SUBAPPLICATION I_GetAttribute_IDA (* Bündelung von I_GetAttribute (Kommando GetAttribute F.58) und Attribute_IDA (asynchroner Adapter-Empfang) mit gemeinsamen u16ObjId und u8AID Parametern *)
  (* Standard: 61499-2; Description: Copyright (c) 2026 Meisterschulen am Ostbahnhof This program and the accompanying materials are made available under the terms of the Eclipse Public License 2.0 which is available at https://www.eclipse.org/legal/epl-2.0/ SPDX-License-Identifier: EPL-2.0 *)
  (* Version 1.0, 2026-09-15, Franz Höpfinger, Meisterschulen am Ostbahnhof, Initial implementation combining I_GetAttribute and Attribute_IDA *)
  PACKAGE isobus::UT::io::Attribute;
  IMPORT isobus::UT::Q::const::IDs::ID_NULL;
  IMPORT isobus::UT::I::I_GetAttribute;
  IMPORT isobus::UT::io::Attribute::Attribute_IDA;
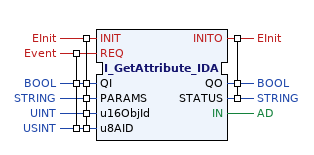
  EVENT_INPUT
    INIT : EInit WITH u16ObjId, u8AID, QI, PARAMS; (* Service Initialization *)
    REQ WITH u8AID, QI; (* Service Request *)
  END_EVENT
  EVENT_OUTPUT
    INITO : EInit WITH QO, STATUS; (* Initialization Confirm *)
  END_EVENT
  VAR_INPUT
    QI : BOOL := TRUE; (* Event Input Qualifier *)
    PARAMS : STRING; (* Service Parameters *)
    u16ObjId : UINT := ID_NULL; (* Object ID *)
    u8AID : USINT; (* Attribute ID of the object *)
  END_VAR
  VAR_OUTPUT
    QO : BOOL; (* Event Output Qualifier *)
    STATUS : STRING; (* Service Status *)
  END_VAR
  PLUGS
    IN : adapter::types::unidirectional::AD; (* Input data from resource *)
  END_PLUGS
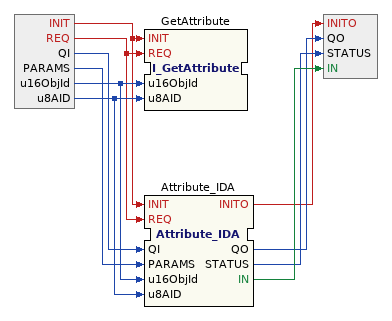
  FBS
    GetAttribute : isobus::UT::I::I_GetAttribute;
    Attribute_IDA : isobus::UT::io::Attribute::Attribute_IDA;
  END_FBS
  EVENT_CONNECTIONS
    INIT TO GetAttribute.INIT;
    INIT TO Attribute_IDA.INIT;
    REQ TO GetAttribute.REQ;
    REQ TO Attribute_IDA.REQ;
    Attribute_IDA.INITO TO INITO;
  END_CONNECTIONS
  DATA_CONNECTIONS
    u16ObjId TO GetAttribute.u16ObjId;
    u16ObjId TO Attribute_IDA.u16ObjId;
    u8AID TO GetAttribute.u8AID;
    u8AID TO Attribute_IDA.u8AID;
    QI TO Attribute_IDA.QI;
    PARAMS TO Attribute_IDA.PARAMS;
    Attribute_IDA.QO TO QO;
    Attribute_IDA.STATUS TO STATUS;
  END_CONNECTIONS
  ADAPTER_CONNECTIONS
    Attribute_IDA.IN TO IN;
  END_CONNECTIONS
END_SUBAPPLICATION
